  650 = 'Clamp Cylinder A1 Failed to Advance... Check Q1.0...' | German: 'S5 650 Row 66 Failed To Advance.. Check Qxxx.x German' | French: 'S5 650 Row 66 Failed To Advance.. Check Qxxx.x French'
  651 = 'Clamp Cylinder A1 Failed to Return... Check Q1.1...' | German: 'S5 651 Row 66 Failed To Return.. Check Qxxx.x German' | French: 'S5 651 Row 66 Failed To Return.. Check Qxxx.x French'
  652 = 'Clamp Cylinder A1 Lost Advanced... Check I1.0...' | German: 'S5 652 Row 66 Lost Advance Position... Check Ixxx.x German' | French: 'S5 652 Row 66 Lost Advance Position... Check Ixxx.x French'
  653 = 'Clamp Cylinder A1 Lost Returned... Check I1.1...' | German: 'S5 653 Row 66 Lost Return Position... Check Ixxx.x German' | French: 'S5 653 Row 66 Lost Return Position... Check Ixxx.x French'
  654 = 'Clamp Cylinder A1 Switch Fault... Check I1.0, I1.1...' | German: 'S5 654 Row 66 Switch Fault... Check Ixxx.x / Ixxx.x German' | French: 'S5 654 Row 66 Switch Fault... Check Ixxx.x / Ixxx.x French'
  655 = 'Spare' | German: 'S5 655 Row 66 Spare Message German' | French: 'S5 655 Row 66 Spare Message French'
  656 = 'Spare' | German: 'S5 656 Row 66 Spare Message German' | French: 'S5 656 Row 66 Spare Message French'
  657 = 'Spare' | German: 'S5 657 Row 66 Spare Message German' | French: 'S5 657 Row 66 Spare Message French'
  658 = 'Spare' | German: 'S5 658 Row 66 Spare Message German' | French: 'S5 658 Row 66 Spare Message French'
  659 = 'Spare' | German: 'S5 659 Row 66 Spare Message German' | French: 'S5 659 Row 66 Spare Message French'
  660 = 'Clamp Cylinder A1 Failed to Advance... Check Q1.0...' | German: 'S5 660 Row 67 Failed To Advance.. Check Qxxx.x German' | French: 'S5 660 Row 67 Failed To Advance.. Check Qxxx.x French'
  661 = 'Clamp Cylinder A1 Failed to Return... Check Q1.1...' | German: 'S5 661 Row 67 Failed To Return.. Check Qxxx.x German' | French: 'S5 661 Row 67 Failed To Return.. Check Qxxx.x French'
  662 = 'Clamp Cylinder A1 Lost Advanced... Check I1.0...' | German: 'S5 662 Row 67 Lost Advance Position... Check Ixxx.x German' | French: 'S5 662 Row 67 Lost Advance Position... Check Ixxx.x French'
  663 = 'Clamp Cylinder A1 Lost Returned... Check I1.1...' | German: 'S5 663 Row 67 Lost Return Position... Check Ixxx.x German' | French: 'S5 663 Row 67 Lost Return Position... Check Ixxx.x French'
  664 = 'Clamp Cylinder A1 Switch Fault... Check I1.0, I1.1...' | German: 'S5 664 Row 67 Switch Fault... Check Ixxx.x / Ixxx.x German' | French: 'S5 664 Row 67 Switch Fault... Check Ixxx.x / Ixxx.x French'
  665 = 'Spare' | German: 'S5 665 Row 67 Spare Message German' | French: 'S5 665 Row 67 Spare Message French'
  666 = 'Spare' | German: 'S5 666 Row 67 Spare Message German' | French: 'S5 666 Row 67 Spare Message French'
  667 = 'Spare' | German: 'S5 667 Row 67 Spare Message German' | French: 'S5 667 Row 67 Spare Message French'
  668 = 'Spare' | German: 'S5 668 Row 67 Spare Message German' | French: 'S5 668 Row 67 Spare Message French'
  669 = 'Spare' | German: 'S5 669 Row 67 Spare Message German' | French: 'S5 669 Row 67 Spare Message French'
  670 = 'Clamp Cylinder A1 Failed to Advance... Check Q1.0...' | German: 'S5 670 Row 68 Failed To Advance.. Check Qxxx.x German' | French: 'S5 670 Row 68 Failed To Advance.. Check Qxxx.x French'
  671 = 'Clamp Cylinder A1 Failed to Return... Check Q1.1...' | German: 'S5 671 Row 68 Failed To Return.. Check Qxxx.x German' | French: 'S5 671 Row 68 Failed To Return.. Check Qxxx.x French'
  672 = 'Clamp Cylinder A1 Lost Advanced... Check I1.0...' | German: 'S5 672 Row 68 Lost Advance Position... Check Ixxx.x German' | French: 'S5 672 Row 68 Lost Advance Position... Check Ixxx.x French'
  673 = 'Clamp Cylinder A1 Lost Returned... Check I1.1...' | German: 'S5 673 Row 68 Lost Return Position... Check Ixxx.x German' | French: 'S5 673 Row 68 Lost Return Position... Check Ixxx.x French'
  674 = 'Clamp Cylinder A1 Switch Fault... Check I1.0, I1.1...' | German: 'S5 674 Row 68 Switch Fault... Check Ixxx.x / Ixxx.x German' | French: 'S5 674 Row 68 Switch Fault... Check Ixxx.x / Ixxx.x French'
  675 = 'Spare' | German: 'S5 675 Row 68 Spare Message German' | French: 'S5 675 Row 68 Spare Message French'
  676 = 'Spare' | German: 'S5 676 Row 68 Spare Message German' | French: 'S5 676 Row 68 Spare Message French'
  677 = 'Spare' | German: 'S5 677 Row 68 Spare Message German' | French: 'S5 677 Row 68 Spare Message French'
  678 = 'Spare' | German: 'S5 678 Row 68 Spare Message German' | French: 'S5 678 Row 68 Spare Message French'
  679 = 'Spare' | German: 'S5 679 Row 68 Spare Message German' | French: 'S5 679 Row 68 Spare Message French'
  680 = 'Clamp Cylinder A1 Failed to Advance... Check Q1.0...' | German: 'S5 680 Row 69 Failed To Advance.. Check Qxxx.x German' | French: 'S5 680 Row 69 Failed To Advance.. Check Qxxx.x French'
  681 = 'Clamp Cylinder A1 Failed to Return... Check Q1.1...' | German: 'S5 681 Row 69 Failed To Return.. Check Qxxx.x German' | French: 'S5 681 Row 69 Failed To Return.. Check Qxxx.x French'
  682 = 'Clamp Cylinder A1 Lost Advanced... Check I1.0...' | German: 'S5 682 Row 69 Lost Advance Position... Check Ixxx.x German' | French: 'S5 682 Row 69 Lost Advance Position... Check Ixxx.x French'
  683 = 'Clamp Cylinder A1 Lost Returned... Check I1.1...' | German: 'S5 683 Row 69 Lost Return Position... Check Ixxx.x German' | French: 'S5 683 Row 69 Lost Return Position... Check Ixxx.x French'
  684 = 'Clamp Cylinder A1 Switch Fault... Check I1.0, I1.1...' | German: 'S5 684 Row 69 Switch Fault... Check Ixxx.x / Ixxx.x German' | French: 'S5 684 Row 69 Switch Fault... Check Ixxx.x / Ixxx.x French'
  685 = 'Spare' | German: 'S5 685 Row 69 Spare Message German' | French: 'S5 685 Row 69 Spare Message French'
  686 = 'Spare' | German: 'S5 686 Row 69 Spare Message German' | French: 'S5 686 Row 69 Spare Message French'
  687 = 'Spare' | German: 'S5 687 Row 69 Spare Message German' | French: 'S5 687 Row 69 Spare Message French'
  688 = 'Spare' | German: 'S5 688 Row 69 Spare Message German' | French: 'S5 688 Row 69 Spare Message French'
  689 = 'Spare' | German: 'S5 689 Row 69 Spare Message German' | French: 'S5 689 Row 69 Spare Message French'
  690 = 'Clamp Cylinder A1 Failed to Advance... Check Q1.0...' | German: 'S5 690 Row 70 Failed To Advance.. Check Qxxx.x German' | French: 'S5 690 Row 70 Failed To Advance.. Check Qxxx.x French'
  691 = 'Clamp Cylinder A1 Failed to Return... Check Q1.1...' | German: 'S5 691 Row 70 Failed To Return.. Check Qxxx.x German' | French: 'S5 691 Row 70 Failed To Return.. Check Qxxx.x French'
  692 = 'Clamp Cylinder A1 Lost Advanced... Check I1.0...' | German: 'S5 692 Row 70 Lost Advance Position... Check Ixxx.x German' | French: 'S5 692 Row 70 Lost Advance Position... Check Ixxx.x French'
  693 = 'Clamp Cylinder A1 Lost Returned... Check I1.1...' | German: 'S5 693 Row 70 Lost Return Position... Check Ixxx.x German' | French: 'S5 693 Row 70 Lost Return Position... Check Ixxx.x French'
  694 = 'Clamp Cylinder A1 Switch Fault... Check I1.0, I1.1...' | German: 'S5 694 Row 70 Switch Fault... Check Ixxx.x / Ixxx.x German' | French: 'S5 694 Row 70 Switch Fault... Check Ixxx.x / Ixxx.x French'
  695 = 'Spare' | German: 'S5 695 Row 70 Spare Message German' | French: 'S5 695 Row 70 Spare Message French'
  696 = 'Spare' | German: 'S5 696 Row 70 Spare Message German' | French: 'S5 696 Row 70 Spare Message French'
  697 = 'Spare' | German: 'S5 697 Row 70 Spare Message German' | French: 'S5 697 Row 70 Spare Message French'
  698 = 'Spare' | German: 'S5 698 Row 70 Spare Message German' | French: 'S5 698 Row 70 Spare Message French'
  699 = 'Spare' | German: 'S5 699 Row 70 Spare Message German' | French: 'S5 699 Row 70 Spare Message French'
  700 = 'Clamp Cylinder A1 Failed to Advance... Check Q1.0...' | German: 'S5 700 Row 71 Failed To Advance.. Check Qxxx.x German' | French: 'S5 700 Row 71 Failed To Advance.. Check Qxxx.x French'
  701 = 'Clamp Cylinder A1 Failed to Return... Check Q1.1...' | German: 'S5 701 Row 71 Failed To Return.. Check Qxxx.x German' | French: 'S5 701 Row 71 Failed To Return.. Check Qxxx.x French'
  702 = 'Clamp Cylinder A1 Lost Advanced... Check I1.0...' | German: 'S5 702 Row 71 Lost Advance Position... Check Ixxx.x German' | French: 'S5 702 Row 71 Lost Advance Position... Check Ixxx.x French'
  703 = 'Clamp Cylinder A1 Lost Returned... Check I1.1...' | German: 'S5 703 Row 71 Lost Return Position... Check Ixxx.x German' | French: 'S5 703 Row 71 Lost Return Position... Check Ixxx.x French'
  704 = 'Clamp Cylinder A1 Switch Fault... Check I1.0, I1.1...' | German: 'S5 704 Row 71 Switch Fault... Check Ixxx.x / Ixxx.x German' | French: 'S5 704 Row 71 Switch Fault... Check Ixxx.x / Ixxx.x French'
  705 = 'Spare' | German: 'S5 705 Row 71 Spare Message German' | French: 'S5 705 Row 71 Spare Message French'
  706 = 'Spare' | German: 'S5 706 Row 71 Spare Message German' | French: 'S5 706 Row 71 Spare Message French'
  707 = 'Spare' | German: 'S5 707 Row 71 Spare Message German' | French: 'S5 707 Row 71 Spare Message French'
  708 = 'Spare' | German: 'S5 708 Row 71 Spare Message German' | French: 'S5 708 Row 71 Spare Message French'
  709 = 'Spare' | German: 'S5 709 Row 71 Spare Message German' | French: 'S5 709 Row 71 Spare Message French'
  710 = 'Clamp Cylinder A1 Failed to Advance... Check Q1.0...' | German: 'S5 710 Row 72 Failed To Advance.. Check Qxxx.x German' | French: 'S5 710 Row 72 Failed To Advance.. Check Qxxx.x French'
  711 = 'Clamp Cylinder A1 Failed to Return... Check Q1.1...' | German: 'S5 711 Row 72 Failed To Return.. Check Qxxx.x German' | French: 'S5 711 Row 72 Failed To Return.. Check Qxxx.x French'
  712 = 'Clamp Cylinder A1 Lost Advanced... Check I1.0...' | German: 'S5 712 Row 72 Lost Advance Position... Check Ixxx.x German' | French: 'S5 712 Row 72 Lost Advance Position... Check Ixxx.x French'
  713 = 'Clamp Cylinder A1 Lost Returned... Check I1.1...' | German: 'S5 713 Row 72 Lost Return Position... Check Ixxx.x German' | French: 'S5 713 Row 72 Lost Return Position... Check Ixxx.x French'
  714 = 'Clamp Cylinder A1 Switch Fault... Check I1.0, I1.1...' | German: 'S5 714 Row 72 Switch Fault... Check Ixxx.x / Ixxx.x German' | French: 'S5 714 Row 72 Switch Fault... Check Ixxx.x / Ixxx.x French'
  715 = 'Spare' | German: 'S5 715 Row 72 Spare Message German' | French: 'S5 715 Row 72 Spare Message French'
  716 = 'Spare' | German: 'S5 716 Row 72 Spare Message German' | French: 'S5 716 Row 72 Spare Message French'
  717 = 'Spare' | German: 'S5 717 Row 72 Spare Message German' | French: 'S5 717 Row 72 Spare Message French'
  718 = 'Spare' | German: 'S5 718 Row 72 Spare Message German' | French: 'S5 718 Row 72 Spare Message French'
  719 = 'Spare' | German: 'S5 719 Row 72 Spare Message German' | French: 'S5 719 Row 72 Spare Message French'
  720 = 'Clamp Cylinder A1 Failed to Advance... Check Q1.0...' | German: 'S5 720 Row 73 Failed To Advance.. Check Qxxx.x German' | French: 'S5 720 Row 73 Failed To Advance.. Check Qxxx.x French'
  721 = 'Clamp Cylinder A1 Failed to Return... Check Q1.1...' | German: 'S5 721 Row 73 Failed To Return.. Check Qxxx.x German' | French: 'S5 721 Row 73 Failed To Return.. Check Qxxx.x French'
  722 = 'Clamp Cylinder A1 Lost Advanced... Check I1.0...' | German: 'S5 722 Row 73 Lost Advance Position... Check Ixxx.x German' | French: 'S5 722 Row 73 Lost Advance Position... Check Ixxx.x French'
  723 = 'Clamp Cylinder A1 Lost Returned... Check I1.1...' | German: 'S5 723 Row 73 Lost Return Position... Check Ixxx.x German' | French: 'S5 723 Row 73 Lost Return Position... Check Ixxx.x French'
  724 = 'Clamp Cylinder A1 Switch Fault... Check I1.0, I1.1...' | German: 'S5 724 Row 73 Switch Fault... Check Ixxx.x / Ixxx.x German' | French: 'S5 724 Row 73 Switch Fault... Check Ixxx.x / Ixxx.x French'
  725 = 'Spare' | German: 'S5 725 Row 73 Spare Message German' | French: 'S5 725 Row 73 Spare Message French'
  726 = 'Spare' | German: 'S5 726 Row 73 Spare Message German' | French: 'S5 726 Row 73 Spare Message French'
  727 = 'Spare' | German: 'S5 727 Row 73 Spare Message German' | French: 'S5 727 Row 73 Spare Message French'
  728 = 'Spare' | German: 'S5 728 Row 73 Spare Message German' | French: 'S5 728 Row 73 Spare Message French'
  729 = 'Spare' | German: 'S5 729 Row 73 Spare Message German' | French: 'S5 729 Row 73 Spare Message French'
  730 = 'Clamp Cylinder A1 Failed to Advance... Check Q1.0...' | German: 'S5 730 Row 74 Failed To Advance.. Check Qxxx.x German' | French: 'S5 730 Row 74 Failed To Advance.. Check Qxxx.x French'
  731 = 'Clamp Cylinder A1 Failed to Return... Check Q1.1...' | German: 'S5 731 Row 74 Failed To Return.. Check Qxxx.x German' | French: 'S5 731 Row 74 Failed To Return.. Check Qxxx.x French'
  732 = 'Clamp Cylinder A1 Lost Advanced... Check I1.0...' | German: 'S5 732 Row 74 Lost Advance Position... Check Ixxx.x German' | French: 'S5 732 Row 74 Lost Advance Position... Check Ixxx.x French'
  733 = 'Clamp Cylinder A1 Lost Returned... Check I1.1...' | German: 'S5 733 Row 74 Lost Return Position... Check Ixxx.x German' | French: 'S5 733 Row 74 Lost Return Position... Check Ixxx.x French'
  734 = 'Clamp Cylinder A1 Switch Fault... Check I1.0, I1.1...' | German: 'S5 734 Row 74 Switch Fault... Check Ixxx.x / Ixxx.x German' | French: 'S5 734 Row 74 Switch Fault... Check Ixxx.x / Ixxx.x French'
  735 = 'Spare' | German: 'S5 735 Row 74 Spare Message German' | French: 'S5 735 Row 74 Spare Message French'
  736 = 'Spare' | German: 'S5 736 Row 74 Spare Message German' | French: 'S5 736 Row 74 Spare Message French'
  737 = 'Spare' | German: 'S5 737 Row 74 Spare Message German' | French: 'S5 737 Row 74 Spare Message French'
  738 = 'Spare' | German: 'S5 738 Row 74 Spare Message German' | French: 'S5 738 Row 74 Spare Message French'
  739 = 'Spare' | German: 'S5 739 Row 74 Spare Message German' | French: 'S5 739 Row 74 Spare Message French'
  740 = 'Clamp Cylinder A1 Failed to Advance... Check Q1.0...' | German: 'S5 740 Row 75 Failed To Advance.. Check Qxxx.x German' | French: 'S5 740 Row 75 Failed To Advance.. Check Qxxx.x French'
  741 = 'Clamp Cylinder A1 Failed to Return... Check Q1.1...' | German: 'S5 741 Row 75 Failed To Return.. Check Qxxx.x German' | French: 'S5 741 Row 75 Failed To Return.. Check Qxxx.x French'
  742 = 'Clamp Cylinder A1 Lost Advanced... Check I1.0...' | German: 'S5 742 Row 75 Lost Advance Position... Check Ixxx.x German' | French: 'S5 742 Row 75 Lost Advance Position... Check Ixxx.x French'
  743 = 'Clamp Cylinder A1 Lost Returned... Check I1.1...' | German: 'S5 743 Row 75 Lost Return Position... Check Ixxx.x German' | French: 'S5 743 Row 75 Lost Return Position... Check Ixxx.x French'
  744 = 'Clamp Cylinder A1 Switch Fault... Check I1.0, I1.1...' | German: 'S5 744 Row 75 Switch Fault... Check Ixxx.x / Ixxx.x German' | French: 'S5 744 Row 75 Switch Fault... Check Ixxx.x / Ixxx.x French'
  745 = 'Spare' | German: 'S5 745 Row 75 Spare Message German' | French: 'S5 745 Row 75 Spare Message French'
  746 = 'Spare' | German: 'S5 746 Row 75 Spare Message German' | French: 'S5 746 Row 75 Spare Message French'
  747 = 'Spare' | German: 'S5 747 Row 75 Spare Message German' | French: 'S5 747 Row 75 Spare Message French'
  748 = 'Spare' | German: 'S5 748 Row 75 Spare Message German' | French: 'S5 748 Row 75 Spare Message French'
  749 = 'Spare' | German: 'S5 749 Row 75 Spare Message German' | French: 'S5 749 Row 75 Spare Message French'
  750 = 'Clamp Cylinder A1 Failed to Advance... Check Q1.0...' | German: 'S5 750 Row 76 Failed To Advance.. Check Qxxx.x German' | French: 'S5 750 Row 76 Failed To Advance.. Check Qxxx.x French'
  751 = 'Clamp Cylinder A1 Failed to Return... Check Q1.1...' | German: 'S5 751 Row 76 Failed To Return.. Check Qxxx.x German' | French: 'S5 751 Row 76 Failed To Return.. Check Qxxx.x French'
  752 = 'Clamp Cylinder A1 Lost Advanced... Check I1.0...' | German: 'S5 752 Row 76 Lost Advance Position... Check Ixxx.x German' | French: 'S5 752 Row 76 Lost Advance Position... Check Ixxx.x French'
  753 = 'Clamp Cylinder A1 Lost Returned... Check I1.1...' | German: 'S5 753 Row 76 Lost Return Position... Check Ixxx.x German' | French: 'S5 753 Row 76 Lost Return Position... Check Ixxx.x French'
  754 = 'Clamp Cylinder A1 Switch Fault... Check I1.0, I1.1...' | German: 'S5 754 Row 76 Switch Fault... Check Ixxx.x / Ixxx.x German' | French: 'S5 754 Row 76 Switch Fault... Check Ixxx.x / Ixxx.x French'
  755 = 'Spare' | German: 'S5 755 Row 76 Spare Message German' | French: 'S5 755 Row 76 Spare Message French'
  756 = 'Spare' | German: 'S5 756 Row 76 Spare Message German' | French: 'S5 756 Row 76 Spare Message French'
  757 = 'Spare' | German: 'S5 757 Row 76 Spare Message German' | French: 'S5 757 Row 76 Spare Message French'
  758 = 'Spare' | German: 'S5 758 Row 76 Spare Message German' | French: 'S5 758 Row 76 Spare Message French'
  759 = 'Spare' | German: 'S5 759 Row 76 Spare Message German' | French: 'S5 759 Row 76 Spare Message French'
  760 = 'Clamp Cylinder A1 Failed to Advance... Check Q1.0...' | German: 'S5 760 Row 77 Failed To Advance.. Check Qxxx.x German' | French: 'S5 760 Row 77 Failed To Advance.. Check Qxxx.x French'
  761 = 'Clamp Cylinder A1 Failed to Return... Check Q1.1...' | German: 'S5 761 Row 77 Failed To Return.. Check Qxxx.x German' | French: 'S5 761 Row 77 Failed To Return.. Check Qxxx.x French'
  762 = 'Clamp Cylinder A1 Lost Advanced... Check I1.0...' | German: 'S5 762 Row 77 Lost Advance Position... Check Ixxx.x German' | French: 'S5 762 Row 77 Lost Advance Position... Check Ixxx.x French'
  763 = 'Clamp Cylinder A1 Lost Returned... Check I1.1...' | German: 'S5 763 Row 77 Lost Return Position... Check Ixxx.x German' | French: 'S5 763 Row 77 Lost Return Position... Check Ixxx.x French'
  764 = 'Clamp Cylinder A1 Switch Fault... Check I1.0, I1.1...' | German: 'S5 764 Row 77 Switch Fault... Check Ixxx.x / Ixxx.x German' | French: 'S5 764 Row 77 Switch Fault... Check Ixxx.x / Ixxx.x French'
  765 = 'Spare' | German: 'S5 765 Row 77 Spare Message German' | French: 'S5 765 Row 77 Spare Message French'
  766 = 'Spare' | German: 'S5 766 Row 77 Spare Message German' | French: 'S5 766 Row 77 Spare Message French'
  767 = 'Spare' | German: 'S5 767 Row 77 Spare Message German' | French: 'S5 767 Row 77 Spare Message French'
  768 = 'Spare' | German: 'S5 768 Row 77 Spare Message German' | French: 'S5 768 Row 77 Spare Message French'
  769 = 'Spare' | German: 'S5 769 Row 77 Spare Message German' | French: 'S5 769 Row 77 Spare Message French'
  770 = 'Clamp Cylinder A1 Failed to Advance... Check Q1.0...' | German: 'S5 770 Row 78 Failed To Advance.. Check Qxxx.x German' | French: 'S5 770 Row 78 Failed To Advance.. Check Qxxx.x French'
  771 = 'Clamp Cylinder A1 Failed to Return... Check Q1.1...' | German: 'S5 771 Row 78 Failed To Return.. Check Qxxx.x German' | French: 'S5 771 Row 78 Failed To Return.. Check Qxxx.x French'
  772 = 'Clamp Cylinder A1 Lost Advanced... Check I1.0...' | German: 'S5 772 Row 78 Lost Advance Position... Check Ixxx.x German' | French: 'S5 772 Row 78 Lost Advance Position... Check Ixxx.x French'
  773 = 'Clamp Cylinder A1 Lost Returned... Check I1.1...' | German: 'S5 773 Row 78 Lost Return Position... Check Ixxx.x German' | French: 'S5 773 Row 78 Lost Return Position... Check Ixxx.x French'
  774 = 'Clamp Cylinder A1 Switch Fault... Check I1.0, I1.1...' | German: 'S5 774 Row 78 Switch Fault... Check Ixxx.x / Ixxx.x German' | French: 'S5 774 Row 78 Switch Fault... Check Ixxx.x / Ixxx.x French'
  775 = 'Spare' | German: 'S5 775 Row 78 Spare Message German' | French: 'S5 775 Row 78 Spare Message French'
  776 = 'Spare' | German: 'S5 776 Row 78 Spare Message German' | French: 'S5 776 Row 78 Spare Message French'
  777 = 'Spare' | German: 'S5 777 Row 78 Spare Message German' | French: 'S5 777 Row 78 Spare Message French'
  778 = 'Spare' | German: 'S5 778 Row 78 Spare Message German' | French: 'S5 778 Row 78 Spare Message French'
  779 = 'Spare' | German: 'S5 779 Row 78 Spare Message German' | French: 'S5 779 Row 78 Spare Message French'
  780 = 'Clamp Cylinder A1 Failed to Advance... Check Q1.0...' | German: 'S5 780 Row 79 Failed To Advance.. Check Qxxx.x German' | French: 'S5 780 Row 79 Failed To Advance.. Check Qxxx.x French'
  781 = 'Clamp Cylinder A1 Failed to Return... Check Q1.1...' | German: 'S5 781 Row 79 Failed To Return.. Check Qxxx.x German' | French: 'S5 781 Row 79 Failed To Return.. Check Qxxx.x French'
  782 = 'Clamp Cylinder A1 Lost Advanced... Check I1.0...' | German: 'S5 782 Row 79 Lost Advance Position... Check Ixxx.x German' | French: 'S5 782 Row 79 Lost Advance Position... Check Ixxx.x French'
  783 = 'Clamp Cylinder A1 Lost Returned... Check I1.1...' | German: 'S5 783 Row 79 Lost Return Position... Check Ixxx.x German' | French: 'S5 783 Row 79 Lost Return Position... Check Ixxx.x French'
  784 = 'Clamp Cylinder A1 Switch Fault... Check I1.0, I1.1...' | German: 'S5 784 Row 79 Switch Fault... Check Ixxx.x / Ixxx.x German' | French: 'S5 784 Row 79 Switch Fault... Check Ixxx.x / Ixxx.x French'
  785 = 'Spare' | German: 'S5 785 Row 79 Spare Message German' | French: 'S5 785 Row 79 Spare Message French'
  786 = 'Spare' | German: 'S5 786 Row 79 Spare Message German' | French: 'S5 786 Row 79 Spare Message French'
  787 = 'Spare' | German: 'S5 787 Row 79 Spare Message German' | French: 'S5 787 Row 79 Spare Message French'
  788 = 'Spare' | German: 'S5 788 Row 79 Spare Message German' | French: 'S5 788 Row 79 Spare Message French'
  789 = 'Spare' | German: 'S5 789 Row 79 Spare Message German' | French: 'S5 789 Row 79 Spare Message French'
  790 = 'Clamp Cylinder A1 Failed to Advance... Check Q1.0...' | German: 'S5 790 Row 80 Failed To Advance.. Check Qxxx.x German' | French: 'S5 790 Row 80 Failed To Advance.. Check Qxxx.x French'
  791 = 'Clamp Cylinder A1 Failed to Return... Check Q1.1...' | German: 'S5 791 Row 80 Failed To Return.. Check Qxxx.x German' | French: 'S5 791 Row 80 Failed To Return.. Check Qxxx.x French'
  792 = 'Clamp Cylinder A1 Lost Advanced... Check I1.0...' | German: 'S5 792 Row 80 Lost Advance Position... Check Ixxx.x German' | French: 'S5 792 Row 80 Lost Advance Position... Check Ixxx.x French'
  793 = 'Clamp Cylinder A1 Lost Returned... Check I1.1...' | German: 'S5 793 Row 80 Lost Return Position... Check Ixxx.x German' | French: 'S5 793 Row 80 Lost Return Position... Check Ixxx.x French'
  794 = 'Clamp Cylinder A1 Switch Fault... Check I1.0, I1.1...' | German: 'S5 794 Row 80 Switch Fault... Check Ixxx.x / Ixxx.x German' | French: 'S5 794 Row 80 Switch Fault... Check Ixxx.x / Ixxx.x French'
  795 = 'Spare' | German: 'S5 795 Row 80 Spare Message German' | French: 'S5 795 Row 80 Spare Message French'
  796 = 'Spare' | German: 'S5 796 Row 80 Spare Message German' | French: 'S5 796 Row 80 Spare Message French'
  797 = 'Spare' | German: 'S5 797 Row 80 Spare Message German' | French: 'S5 797 Row 80 Spare Message French'
  798 = 'Spare' | German: 'S5 798 Row 80 Spare Message German' | French: 'S5 798 Row 80 Spare Message French'
  799 = 'Spare' | German: 'S5 799 Row 80 Spare Message German' | French: 'S5 799 Row 80 Spare Message French'
  800 = 'Clamp Cylinder A1 Failed to Advance... Check Q1.0...' | German: 'S5 800 Row 81 Failed To Advance.. Check Qxxx.x German' | French: 'S5 800 Row 81 Failed To Advance.. Check Qxxx.x French'
  801 = 'Clamp Cylinder A1 Failed to Return... Check Q1.1...' | German: 'S5 801 Row 81 Failed To Return.. Check Qxxx.x German' | French: 'S5 801 Row 81 Failed To Return.. Check Qxxx.x French'
  802 = 'Clamp Cylinder A1 Lost Advanced... Check I1.0...' | German: 'S5 802 Row 81 Lost Advance Position... Check Ixxx.x German' | French: 'S5 802 Row 81 Lost Advance Position... Check Ixxx.x French'
  803 = 'Clamp Cylinder A1 Lost Returned... Check I1.1...' | German: 'S5 803 Row 81 Lost Return Position... Check Ixxx.x German' | French: 'S5 803 Row 81 Lost Return Position... Check Ixxx.x French'
  804 = 'Clamp Cylinder A1 Switch Fault... Check I1.0, I1.1...' | German: 'S5 804 Row 81 Switch Fault... Check Ixxx.x / Ixxx.x German' | French: 'S5 804 Row 81 Switch Fault... Check Ixxx.x / Ixxx.x French'
  805 = 'Spare' | German: 'S5 805 Row 81 Spare Message German' | French: 'S5 805 Row 81 Spare Message French'
  806 = 'Spare' | German: 'S5 806 Row 81 Spare Message German' | French: 'S5 806 Row 81 Spare Message French'
  807 = 'Spare' | German: 'S5 807 Row 81 Spare Message German' | French: 'S5 807 Row 81 Spare Message French'
  808 = 'Spare' | German: 'S5 808 Row 81 Spare Message German' | French: 'S5 808 Row 81 Spare Message French'
  809 = 'Spare' | German: 'S5 809 Row 81 Spare Message German' | French: 'S5 809 Row 81 Spare Message French'
  810 = 'Clamp Cylinder A1 Failed to Advance... Check Q1.0...' | German: 'S5 810 Row 82 Failed To Advance.. Check Qxxx.x German' | French: 'S5 810 Row 82 Failed To Advance.. Check Qxxx.x French'
  811 = 'Clamp Cylinder A1 Failed to Return... Check Q1.1...' | German: 'S5 811 Row 82 Failed To Return.. Check Qxxx.x German' | French: 'S5 811 Row 82 Failed To Return.. Check Qxxx.x French'
  812 = 'Clamp Cylinder A1 Lost Advanced... Check I1.0...' | German: 'S5 812 Row 82 Lost Advance Position... Check Ixxx.x German' | French: 'S5 812 Row 82 Lost Advance Position... Check Ixxx.x French'
  813 = 'Clamp Cylinder A1 Lost Returned... Check I1.1...' | German: 'S5 813 Row 82 Lost Return Position... Check Ixxx.x German' | French: 'S5 813 Row 82 Lost Return Position... Check Ixxx.x French'
  814 = 'Clamp Cylinder A1 Switch Fault... Check I1.0, I1.1...' | German: 'S5 814 Row 82 Switch Fault... Check Ixxx.x / Ixxx.x German' | French: 'S5 814 Row 82 Switch Fault... Check Ixxx.x / Ixxx.x French'
  815 = 'Spare' | German: 'S5 815 Row 82 Spare Message German' | French: 'S5 815 Row 82 Spare Message French'
  816 = 'Spare' | German: 'S5 816 Row 82 Spare Message German' | French: 'S5 816 Row 82 Spare Message French'
  817 = 'Spare' | German: 'S5 817 Row 82 Spare Message German' | French: 'S5 817 Row 82 Spare Message French'
  818 = 'Spare' | German: 'S5 818 Row 82 Spare Message German' | French: 'S5 818 Row 82 Spare Message French'
  819 = 'Spare' | German: 'S5 819 Row 82 Spare Message German' | French: 'S5 819 Row 82 Spare Message French'
  820 = 'Clamp Cylinder A1 Failed to Advance... Check Q1.0...' | German: 'S5 820 Row 83 Failed To Advance.. Check Qxxx.x German' | French: 'S5 820 Row 83 Failed To Advance.. Check Qxxx.x French'
  821 = 'Clamp Cylinder A1 Failed to Return... Check Q1.1...' | German: 'S5 821 Row 83 Failed To Return.. Check Qxxx.x German' | French: 'S5 821 Row 83 Failed To Return.. Check Qxxx.x French'
  822 = 'Clamp Cylinder A1 Lost Advanced... Check I1.0...' | German: 'S5 822 Row 83 Lost Advance Position... Check Ixxx.x German' | French: 'S5 822 Row 83 Lost Advance Position... Check Ixxx.x French'
  823 = 'Clamp Cylinder A1 Lost Returned... Check I1.1...' | German: 'S5 823 Row 83 Lost Return Position... Check Ixxx.x German' | French: 'S5 823 Row 83 Lost Return Position... Check Ixxx.x French'
  824 = 'Clamp Cylinder A1 Switch Fault... Check I1.0, I1.1...' | German: 'S5 824 Row 83 Switch Fault... Check Ixxx.x / Ixxx.x German' | French: 'S5 824 Row 83 Switch Fault... Check Ixxx.x / Ixxx.x French'
  825 = 'Spare' | German: 'S5 825 Row 83 Spare Message German' | French: 'S5 825 Row 83 Spare Message French'
  826 = 'Spare' | German: 'S5 826 Row 83 Spare Message German' | French: 'S5 826 Row 83 Spare Message French'
  827 = 'Spare' | German: 'S5 827 Row 83 Spare Message German' | French: 'S5 827 Row 83 Spare Message French'
  828 = 'Spare' | German: 'S5 828 Row 83 Spare Message German' | French: 'S5 828 Row 83 Spare Message French'
  829 = 'Spare' | German: 'S5 829 Row 83 Spare Message German' | French: 'S5 829 Row 83 Spare Message French'
  830 = 'Clamp Cylinder A1 Failed to Advance... Check Q1.0...' | German: 'S5 830 Row 84 Failed To Advance.. Check Qxxx.x German' | French: 'S5 830 Row 84 Failed To Advance.. Check Qxxx.x French'
  831 = 'Clamp Cylinder A1 Failed to Return... Check Q1.1...' | German: 'S5 831 Row 84 Failed To Return.. Check Qxxx.x German' | French: 'S5 831 Row 84 Failed To Return.. Check Qxxx.x French'
  832 = 'Clamp Cylinder A1 Lost Advanced... Check I1.0...' | German: 'S5 832 Row 84 Lost Advance Position... Check Ixxx.x German' | French: 'S5 832 Row 84 Lost Advance Position... Check Ixxx.x French'
  833 = 'Clamp Cylinder A1 Lost Returned... Check I1.1...' | German: 'S5 833 Row 84 Lost Return Position... Check Ixxx.x German' | French: 'S5 833 Row 84 Lost Return Position... Check Ixxx.x French'
  834 = 'Clamp Cylinder A1 Switch Fault... Check I1.0, I1.1...' | German: 'S5 834 Row 84 Switch Fault... Check Ixxx.x / Ixxx.x German' | French: 'S5 834 Row 84 Switch Fault... Check Ixxx.x / Ixxx.x French'
  835 = 'Spare' | German: 'S5 835 Row 84 Spare Message German' | French: 'S5 835 Row 84 Spare Message French'
  836 = 'Spare' | German: 'S5 836 Row 84 Spare Message German' | French: 'S5 836 Row 84 Spare Message French'
  837 = 'Spare' | German: 'S5 837 Row 84 Spare Message German' | French: 'S5 837 Row 84 Spare Message French'
  838 = 'Spare' | German: 'S5 838 Row 84 Spare Message German' | French: 'S5 838 Row 84 Spare Message French'
  839 = 'Spare' | German: 'S5 839 Row 84 Spare Message German' | French: 'S5 839 Row 84 Spare Message French'
  840 = 'Clamp Cylinder A1 Failed to Advance... Check Q1.0...' | German: 'S5 840 Row 85 Failed To Advance.. Check Qxxx.x German' | French: 'S5 840 Row 85 Failed To Advance.. Check Qxxx.x French'
  841 = 'Clamp Cylinder A1 Failed to Return... Check Q1.1...' | German: 'S5 841 Row 85 Failed To Return.. Check Qxxx.x German' | French: 'S5 841 Row 85 Failed To Return.. Check Qxxx.x French'
  842 = 'Clamp Cylinder A1 Lost Advanced... Check I1.0...' | German: 'S5 842 Row 85 Lost Advance Position... Check Ixxx.x German' | French: 'S5 842 Row 85 Lost Advance Position... Check Ixxx.x French'
  843 = 'Clamp Cylinder A1 Lost Returned... Check I1.1...' | German: 'S5 843 Row 85 Lost Return Position... Check Ixxx.x German' | French: 'S5 843 Row 85 Lost Return Position... Check Ixxx.x French'
  844 = 'Clamp Cylinder A1 Switch Fault... Check I1.0, I1.1...' | German: 'S5 844 Row 85 Switch Fault... Check Ixxx.x / Ixxx.x German' | French: 'S5 844 Row 85 Switch Fault... Check Ixxx.x / Ixxx.x French'
  845 = 'Spare' | German: 'S5 845 Row 85 Spare Message German' | French: 'S5 845 Row 85 Spare Message French'
  846 = 'Spare' | German: 'S5 846 Row 85 Spare Message German' | French: 'S5 846 Row 85 Spare Message French'
  847 = 'Spare' | German: 'S5 847 Row 85 Spare Message German' | French: 'S5 847 Row 85 Spare Message French'
  848 = 'Spare' | German: 'S5 848 Row 85 Spare Message German' | French: 'S5 848 Row 85 Spare Message French'
  849 = 'Spare' | German: 'S5 849 Row 85 Spare Message German' | French: 'S5 849 Row 85 Spare Message French'
  850 = 'Clamp Cylinder A1 Failed to Advance... Check Q1.0...' | German: 'S5 850 Row 86 Failed To Advance.. Check Qxxx.x German' | French: 'S5 850 Row 86 Failed To Advance.. Check Qxxx.x French'
  851 = 'Clamp Cylinder A1 Failed to Return... Check Q1.1...' | German: 'S5 851 Row 86 Failed To Return.. Check Qxxx.x German' | French: 'S5 851 Row 86 Failed To Return.. Check Qxxx.x French'
  852 = 'Clamp Cylinder A1 Lost Advanced... Check I1.0...' | German: 'S5 852 Row 86 Lost Advance Position... Check Ixxx.x German' | French: 'S5 852 Row 86 Lost Advance Position... Check Ixxx.x French'
  853 = 'Clamp Cylinder A1 Lost Returned... Check I1.1...' | German: 'S5 853 Row 86 Lost Return Position... Check Ixxx.x German' | French: 'S5 853 Row 86 Lost Return Position... Check Ixxx.x French'
  854 = 'Clamp Cylinder A1 Switch Fault... Check I1.0, I1.1...' | German: 'S5 854 Row 86 Switch Fault... Check Ixxx.x / Ixxx.x German' | French: 'S5 854 Row 86 Switch Fault... Check Ixxx.x / Ixxx.x French'
  855 = 'Spare' | German: 'S5 855 Row 86 Spare Message German' | French: 'S5 855 Row 86 Spare Message French'
  856 = 'Spare' | German: 'S5 856 Row 86 Spare Message German' | French: 'S5 856 Row 86 Spare Message French'
  857 = 'Spare' | German: 'S5 857 Row 86 Spare Message German' | French: 'S5 857 Row 86 Spare Message French'
  858 = 'Spare' | German: 'S5 858 Row 86 Spare Message German' | French: 'S5 858 Row 86 Spare Message French'
  859 = 'Spare' | German: 'S5 859 Row 86 Spare Message German' | French: 'S5 859 Row 86 Spare Message French'
  860 = 'Clamp Cylinder A1 Failed to Advance... Check Q1.0...' | German: 'S5 860 Row 87 Failed To Advance.. Check Qxxx.x German' | French: 'S5 860 Row 87 Failed To Advance.. Check Qxxx.x French'
  861 = 'Clamp Cylinder A1 Failed to Return... Check Q1.1...' | German: 'S5 861 Row 87 Failed To Return.. Check Qxxx.x German' | French: 'S5 861 Row 87 Failed To Return.. Check Qxxx.x French'
  862 = 'Clamp Cylinder A1 Lost Advanced... Check I1.0...' | German: 'S5 862 Row 87 Lost Advance Position... Check Ixxx.x German' | French: 'S5 862 Row 87 Lost Advance Position... Check Ixxx.x French'
  863 = 'Clamp Cylinder A1 Lost Returned... Check I1.1...' | German: 'S5 863 Row 87 Lost Return Position... Check Ixxx.x German' | French: 'S5 863 Row 87 Lost Return Position... Check Ixxx.x French'
  864 = 'Clamp Cylinder A1 Switch Fault... Check I1.0, I1.1...' | German: 'S5 864 Row 87 Switch Fault... Check Ixxx.x / Ixxx.x German' | French: 'S5 864 Row 87 Switch Fault... Check Ixxx.x / Ixxx.x French'
  865 = 'Spare' | German: 'S5 865 Row 87 Spare Message German' | French: 'S5 865 Row 87 Spare Message French'
  866 = 'Spare' | German: 'S5 866 Row 87 Spare Message German' | French: 'S5 866 Row 87 Spare Message French'
  867 = 'Spare' | German: 'S5 867 Row 87 Spare Message German' | French: 'S5 867 Row 87 Spare Message French'
  868 = 'Spare' | German: 'S5 868 Row 87 Spare Message German' | French: 'S5 868 Row 87 Spare Message French'
  869 = 'Spare' | German: 'S5 869 Row 87 Spare Message German' | French: 'S5 869 Row 87 Spare Message French'
  870 = 'Clamp Cylinder A1 Failed to Advance... Check Q1.0...' | German: 'S5 870 Row 88 Failed To Advance.. Check Qxxx.x German' | French: 'S5 870 Row 88 Failed To Advance.. Check Qxxx.x French'
  871 = 'Clamp Cylinder A1 Failed to Return... Check Q1.1...' | German: 'S5 871 Row 88 Failed To Return.. Check Qxxx.x German' | French: 'S5 871 Row 88 Failed To Return.. Check Qxxx.x French'
  872 = 'Clamp Cylinder A1 Lost Advanced... Check I1.0...' | German: 'S5 872 Row 88 Lost Advance Position... Check Ixxx.x German' | French: 'S5 872 Row 88 Lost Advance Position... Check Ixxx.x French'
  873 = 'Clamp Cylinder A1 Lost Returned... Check I1.1...' | German: 'S5 873 Row 88 Lost Return Position... Check Ixxx.x German' | French: 'S5 873 Row 88 Lost Return Position... Check Ixxx.x French'
  874 = 'Clamp Cylinder A1 Switch Fault... Check I1.0, I1.1...' | German: 'S5 874 Row 88 Switch Fault... Check Ixxx.x / Ixxx.x German' | French: 'S5 874 Row 88 Switch Fault... Check Ixxx.x / Ixxx.x French'
  875 = 'Spare' | German: 'S5 875 Row 88 Spare Message German' | French: 'S5 875 Row 88 Spare Message French'
  876 = 'Spare' | German: 'S5 876 Row 88 Spare Message German' | French: 'S5 876 Row 88 Spare Message French'
  877 = 'Spare' | German: 'S5 877 Row 88 Spare Message German' | French: 'S5 877 Row 88 Spare Message French'
  878 = 'Spare' | German: 'S5 878 Row 88 Spare Message German' | French: 'S5 878 Row 88 Spare Message French'
  879 = 'Spare' | German: 'S5 879 Row 88 Spare Message German' | French: 'S5 879 Row 88 Spare Message French'
  880 = 'Clamp Cylinder A1 Failed to Advance... Check Q1.0...' | German: 'S5 880 Row 89 Failed To Advance.. Check Qxxx.x German' | French: 'S5 880 Row 89 Failed To Advance.. Check Qxxx.x French'
  881 = 'Clamp Cylinder A1 Failed to Return... Check Q1.1...' | German: 'S5 881 Row 89 Failed To Return.. Check Qxxx.x German' | French: 'S5 881 Row 89 Failed To Return.. Check Qxxx.x French'
  882 = 'Clamp Cylinder A1 Lost Advanced... Check I1.0...' | German: 'S5 882 Row 89 Lost Advance Position... Check Ixxx.x German' | French: 'S5 882 Row 89 Lost Advance Position... Check Ixxx.x French'
  883 = 'Clamp Cylinder A1 Lost Returned... Check I1.1...' | German: 'S5 883 Row 89 Lost Return Position... Check Ixxx.x German' | French: 'S5 883 Row 89 Lost Return Position... Check Ixxx.x French'
  884 = 'Clamp Cylinder A1 Switch Fault... Check I1.0, I1.1...' | German: 'S5 884 Row 89 Switch Fault... Check Ixxx.x / Ixxx.x German' | French: 'S5 884 Row 89 Switch Fault... Check Ixxx.x / Ixxx.x French'
  885 = 'Spare' | German: 'S5 885 Row 89 Spare Message German' | French: 'S5 885 Row 89 Spare Message French'
  886 = 'Spare' | German: 'S5 886 Row 89 Spare Message German' | French: 'S5 886 Row 89 Spare Message French'
  887 = 'Spare' | German: 'S5 887 Row 89 Spare Message German' | French: 'S5 887 Row 89 Spare Message French'
  888 = 'Spare' | German: 'S5 888 Row 89 Spare Message German' | French: 'S5 888 Row 89 Spare Message French'
  889 = 'Spare' | German: 'S5 889 Row 89 Spare Message German' | French: 'S5 889 Row 89 Spare Message French'
  890 = 'Clamp Cylinder A1 Failed to Advance... Check Q1.0...' | German: 'S5 890 Row 90 Failed To Advance.. Check Qxxx.x German' | French: 'S5 890 Row 90 Failed To Advance.. Check Qxxx.x French'
  891 = 'Clamp Cylinder A1 Failed to Return... Check Q1.1...' | German: 'S5 891 Row 90 Failed To Return.. Check Qxxx.x German' | French: 'S5 891 Row 90 Failed To Return.. Check Qxxx.x French'
  892 = 'Clamp Cylinder A1 Lost Advanced... Check I1.0...' | German: 'S5 892 Row 90 Lost Advance Position... Check Ixxx.x German' | French: 'S5 892 Row 90 Lost Advance Position... Check Ixxx.x French'
  893 = 'Clamp Cylinder A1 Lost Returned... Check I1.1...' | German: 'S5 893 Row 90 Lost Return Position... Check Ixxx.x German' | French: 'S5 893 Row 90 Lost Return Position... Check Ixxx.x French'
  894 = 'Clamp Cylinder A1 Switch Fault... Check I1.0, I1.1...' | German: 'S5 894 Row 90 Switch Fault... Check Ixxx.x / Ixxx.x German' | French: 'S5 894 Row 90 Switch Fault... Check Ixxx.x / Ixxx.x French'
  895 = 'Spare' | German: 'S5 895 Row 90 Spare Message German' | French: 'S5 895 Row 90 Spare Message French'
  896 = 'Spare' | German: 'S5 896 Row 90 Spare Message German' | French: 'S5 896 Row 90 Spare Message French'
  897 = 'Spare' | German: 'S5 897 Row 90 Spare Message German' | French: 'S5 897 Row 90 Spare Message French'
  898 = 'Spare' | German: 'S5 898 Row 90 Spare Message German' | French: 'S5 898 Row 90 Spare Message French'
  899 = 'Spare' | German: 'S5 899 Row 90 Spare Message German' | French: 'S5 899 Row 90 Spare Message French'
  900 = 'Clamp Cylinder A1 Failed to Advance... Check Q1.0...' | German: 'S5 900 Row 91 Failed To Advance.. Check Qxxx.x German' | French: 'S5 900 Row 91 Failed To Advance.. Check Qxxx.x French'
  901 = 'Clamp Cylinder A1 Failed to Return... Check Q1.1...' | German: 'S5 901 Row 91 Failed To Return.. Check Qxxx.x German' | French: 'S5 901 Row 91 Failed To Return.. Check Qxxx.x French'
  902 = 'Clamp Cylinder A1 Lost Advanced... Check I1.0...' | German: 'S5 902 Row 91 Lost Advance Position... Check Ixxx.x German' | French: 'S5 902 Row 91 Lost Advance Position... Check Ixxx.x French'
  903 = 'Clamp Cylinder A1 Lost Returned... Check I1.1...' | German: 'S5 903 Row 91 Lost Return Position... Check Ixxx.x German' | French: 'S5 903 Row 91 Lost Return Position... Check Ixxx.x French'
  904 = 'Clamp Cylinder A1 Switch Fault... Check I1.0, I1.1...' | German: 'S5 904 Row 91 Switch Fault... Check Ixxx.x / Ixxx.x German' | French: 'S5 904 Row 91 Switch Fault... Check Ixxx.x / Ixxx.x French'
  905 = 'Spare' | German: 'S5 905 Row 91 Spare Message German' | French: 'S5 905 Row 91 Spare Message French'
  906 = 'Spare' | German: 'S5 906 Row 91 Spare Message German' | French: 'S5 906 Row 91 Spare Message French'
  907 = 'Spare' | German: 'S5 907 Row 91 Spare Message German' | French: 'S5 907 Row 91 Spare Message French'
  908 = 'Spare' | German: 'S5 908 Row 91 Spare Message German' | French: 'S5 908 Row 91 Spare Message French'
  909 = 'Spare' | German: 'S5 909 Row 91 Spare Message German' | French: 'S5 909 Row 91 Spare Message French'
  910 = 'Clamp Cylinder A1 Failed to Advance... Check Q1.0...' | German: 'S5 910 Row 92 Failed To Advance.. Check Qxxx.x German' | French: 'S5 910 Row 92 Failed To Advance.. Check Qxxx.x French'
  911 = 'Clamp Cylinder A1 Failed to Return... Check Q1.1...' | German: 'S5 911 Row 92 Failed To Return.. Check Qxxx.x German' | French: 'S5 911 Row 92 Failed To Return.. Check Qxxx.x French'
  912 = 'Clamp Cylinder A1 Lost Advanced... Check I1.0...' | German: 'S5 912 Row 92 Lost Advance Position... Check Ixxx.x German' | French: 'S5 912 Row 92 Lost Advance Position... Check Ixxx.x French'
  913 = 'Clamp Cylinder A1 Lost Returned... Check I1.1...' | German: 'S5 913 Row 92 Lost Return Position... Check Ixxx.x German' | French: 'S5 913 Row 92 Lost Return Position... Check Ixxx.x French'
  914 = 'Clamp Cylinder A1 Switch Fault... Check I1.0, I1.1...' | German: 'S5 914 Row 92 Switch Fault... Check Ixxx.x / Ixxx.x German' | French: 'S5 914 Row 92 Switch Fault... Check Ixxx.x / Ixxx.x French'
  915 = 'Spare' | German: 'S5 915 Row 92 Spare Message German' | French: 'S5 915 Row 92 Spare Message French'
  916 = 'Spare' | German: 'S5 916 Row 92 Spare Message German' | French: 'S5 916 Row 92 Spare Message French'
  917 = 'Spare' | German: 'S5 917 Row 92 Spare Message German' | French: 'S5 917 Row 92 Spare Message French'
  918 = 'Spare' | German: 'S5 918 Row 92 Spare Message German' | French: 'S5 918 Row 92 Spare Message French'
  919 = 'Spare' | German: 'S5 919 Row 92 Spare Message German' | French: 'S5 919 Row 92 Spare Message French'
  920 = 'Clamp Cylinder A1 Failed to Advance... Check Q1.0...' | German: 'S5 920 Row 93 Failed To Advance.. Check Qxxx.x German' | French: 'S5 920 Row 93 Failed To Advance.. Check Qxxx.x French'
  921 = 'Clamp Cylinder A1 Failed to Return... Check Q1.1...' | German: 'S5 921 Row 93 Failed To Return.. Check Qxxx.x German' | French: 'S5 921 Row 93 Failed To Return.. Check Qxxx.x French'
  922 = 'Clamp Cylinder A1 Lost Advanced... Check I1.0...' | German: 'S5 922 Row 93 Lost Advance Position... Check Ixxx.x German' | French: 'S5 922 Row 93 Lost Advance Position... Check Ixxx.x French'
  923 = 'Clamp Cylinder A1 Lost Returned... Check I1.1...' | German: 'S5 923 Row 93 Lost Return Position... Check Ixxx.x German' | French: 'S5 923 Row 93 Lost Return Position... Check Ixxx.x French'
  924 = 'Clamp Cylinder A1 Switch Fault... Check I1.0, I1.1...' | German: 'S5 924 Row 93 Switch Fault... Check Ixxx.x / Ixxx.x German' | French: 'S5 924 Row 93 Switch Fault... Check Ixxx.x / Ixxx.x French'
  925 = 'Spare' | German: 'S5 925 Row 93 Spare Message German' | French: 'S5 925 Row 93 Spare Message French'
  926 = 'Spare' | German: 'S5 926 Row 93 Spare Message German' | French: 'S5 926 Row 93 Spare Message French'
  927 = 'Spare' | German: 'S5 927 Row 93 Spare Message German' | French: 'S5 927 Row 93 Spare Message French'
  928 = 'Spare' | German: 'S5 928 Row 93 Spare Message German' | French: 'S5 928 Row 93 Spare Message French'
  929 = 'Spare' | German: 'S5 929 Row 93 Spare Message German' | French: 'S5 929 Row 93 Spare Message French'
  930 = 'Clamp Cylinder A1 Failed to Advance... Check Q1.0...' | German: 'S5 930 Row 94 Failed To Advance.. Check Qxxx.x German' | French: 'S5 930 Row 94 Failed To Advance.. Check Qxxx.x French'
  931 = 'Clamp Cylinder A1 Failed to Return... Check Q1.1...' | German: 'S5 931 Row 94 Failed To Return.. Check Qxxx.x German' | French: 'S5 931 Row 94 Failed To Return.. Check Qxxx.x French'
  932 = 'Clamp Cylinder A1 Lost Advanced... Check I1.0...' | German: 'S5 932 Row 94 Lost Advance Position... Check Ixxx.x German' | French: 'S5 932 Row 94 Lost Advance Position... Check Ixxx.x French'
  933 = 'Clamp Cylinder A1 Lost Returned... Check I1.1...' | German: 'S5 933 Row 94 Lost Return Position... Check Ixxx.x German' | French: 'S5 933 Row 94 Lost Return Position... Check Ixxx.x French'
  934 = 'Clamp Cylinder A1 Switch Fault... Check I1.0, I1.1...' | German: 'S5 934 Row 94 Switch Fault... Check Ixxx.x / Ixxx.x German' | French: 'S5 934 Row 94 Switch Fault... Check Ixxx.x / Ixxx.x French'
  935 = 'Spare' | German: 'S5 935 Row 94 Spare Message German' | French: 'S5 935 Row 94 Spare Message French'
  936 = 'Spare' | German: 'S5 936 Row 94 Spare Message German' | French: 'S5 936 Row 94 Spare Message French'
  937 = 'Spare' | German: 'S5 937 Row 94 Spare Message German' | French: 'S5 937 Row 94 Spare Message French'
  938 = 'Spare' | German: 'S5 938 Row 94 Spare Message German' | French: 'S5 938 Row 94 Spare Message French'
  939 = 'Spare' | German: 'S5 939 Row 94 Spare Message German' | French: 'S5 939 Row 94 Spare Message French'
  940 = 'Clamp Cylinder A1 Failed to Advance... Check Q1.0...' | German: 'S5 940 Row 95 Failed To Advance.. Check Qxxx.x German' | French: 'S5 940 Row 95 Failed To Advance.. Check Qxxx.x French'
  941 = 'Clamp Cylinder A1 Failed to Return... Check Q1.1...' | German: 'S5 941 Row 95 Failed To Return.. Check Qxxx.x German' | French: 'S5 941 Row 95 Failed To Return.. Check Qxxx.x French'
  942 = 'Clamp Cylinder A1 Lost Advanced... Check I1.0...' | German: 'S5 942 Row 95 Lost Advance Position... Check Ixxx.x German' | French: 'S5 942 Row 95 Lost Advance Position... Check Ixxx.x French'
  943 = 'Clamp Cylinder A1 Lost Returned... Check I1.1...' | German: 'S5 943 Row 95 Lost Return Position... Check Ixxx.x German' | French: 'S5 943 Row 95 Lost Return Position... Check Ixxx.x French'
  944 = 'Clamp Cylinder A1 Switch Fault... Check I1.0, I1.1...' | German: 'S5 944 Row 95 Switch Fault... Check Ixxx.x / Ixxx.x German' | French: 'S5 944 Row 95 Switch Fault... Check Ixxx.x / Ixxx.x French'
  945 = 'Spare' | German: 'S5 945 Row 95 Spare Message German' | French: 'S5 945 Row 95 Spare Message French'
  946 = 'Spare' | German: 'S5 946 Row 95 Spare Message German' | French: 'S5 946 Row 95 Spare Message French'
  947 = 'Spare' | German: 'S5 947 Row 95 Spare Message German' | French: 'S5 947 Row 95 Spare Message French'
  948 = 'Spare' | German: 'S5 948 Row 95 Spare Message German' | French: 'S5 948 Row 95 Spare Message French'
  949 = 'Spare' | German: 'S5 949 Row 95 Spare Message German' | French: 'S5 949 Row 95 Spare Message French'
  950 = 'Clamp Cylinder A1 Failed to Advance... Check Q1.0...' | German: 'S5 950 Row 96 Failed To Advance.. Check Qxxx.x German' | French: 'S5 950 Row 96 Failed To Advance.. Check Qxxx.x French'
  951 = 'Clamp Cylinder A1 Failed to Return... Check Q1.1...' | German: 'S5 951 Row 96 Failed To Return.. Check Qxxx.x German' | French: 'S5 951 Row 96 Failed To Return.. Check Qxxx.x French'
  952 = 'Clamp Cylinder A1 Lost Advanced... Check I1.0...' | German: 'S5 952 Row 96 Lost Advance Position... Check Ixxx.x German' | French: 'S5 952 Row 96 Lost Advance Position... Check Ixxx.x French'
  953 = 'Clamp Cylinder A1 Lost Returned... Check I1.1...' | German: 'S5 953 Row 96 Lost Return Position... Check Ixxx.x German' | French: 'S5 953 Row 96 Lost Return Position... Check Ixxx.x French'
  954 = 'Clamp Cylinder A1 Switch Fault... Check I1.0, I1.1...' | German: 'S5 954 Row 96 Switch Fault... Check Ixxx.x / Ixxx.x German' | French: 'S5 954 Row 96 Switch Fault... Check Ixxx.x / Ixxx.x French'
  955 = 'Spare' | German: 'S5 955 Row 96 Spare Message German' | French: 'S5 955 Row 96 Spare Message French'
  956 = 'Spare' | German: 'S5 956 Row 96 Spare Message German' | French: 'S5 956 Row 96 Spare Message French'
  957 = 'Spare' | German: 'S5 957 Row 96 Spare Message German' | French: 'S5 957 Row 96 Spare Message French'
  958 = 'Spare' | German: 'S5 958 Row 96 Spare Message German' | French: 'S5 958 Row 96 Spare Message French'
  959 = 'Spare' | German: 'S5 959 Row 96 Spare Message German' | French: 'S5 959 Row 96 Spare Message French'
  960 = 'Clamp Cylinder A1 Failed to Advance... Check Q1.0...' | German: 'S5 960 Row 97 Failed To Advance.. Check Qxxx.x German' | French: 'S5 960 Row 97 Failed To Advance.. Check Qxxx.x French'
  961 = 'Clamp Cylinder A1 Failed to Return... Check Q1.1...' | German: 'S5 961 Row 97 Failed To Return.. Check Qxxx.x German' | French: 'S5 961 Row 97 Failed To Return.. Check Qxxx.x French'
  962 = 'Clamp Cylinder A1 Lost Advanced... Check I1.0...' | German: 'S5 962 Row 97 Lost Advance Position... Check Ixxx.x German' | French: 'S5 962 Row 97 Lost Advance Position... Check Ixxx.x French'
  963 = 'Clamp Cylinder A1 Lost Returned... Check I1.1...' | German: 'S5 963 Row 97 Lost Return Position... Check Ixxx.x German' | French: 'S5 963 Row 97 Lost Return Position... Check Ixxx.x French'
  964 = 'Clamp Cylinder A1 Switch Fault... Check I1.0, I1.1...' | German: 'S5 964 Row 97 Switch Fault... Check Ixxx.x / Ixxx.x German' | French: 'S5 964 Row 97 Switch Fault... Check Ixxx.x / Ixxx.x French'
  965 = 'Spare' | German: 'S5 965 Row 97 Spare Message German' | French: 'S5 965 Row 97 Spare Message French'
  966 = 'Spare' | German: 'S5 966 Row 97 Spare Message German' | French: 'S5 966 Row 97 Spare Message French'
  967 = 'Spare' | German: 'S5 967 Row 97 Spare Message German' | French: 'S5 967 Row 97 Spare Message French'
  968 = 'Spare' | German: 'S5 968 Row 97 Spare Message German' | French: 'S5 968 Row 97 Spare Message French'
  969 = 'Spare' | German: 'S5 969 Row 97 Spare Message German' | French: 'S5 969 Row 97 Spare Message French'
  970 = 'Clamp Cylinder A1 Failed to Advance... Check Q1.0...' | German: 'S5 970 Row 98 Failed To Advance.. Check Qxxx.x German' | French: 'S5 970 Row 98 Failed To Advance.. Check Qxxx.x French'
  971 = 'Clamp Cylinder A1 Failed to Return... Check Q1.1...' | German: 'S5 971 Row 98 Failed To Return.. Check Qxxx.x German' | French: 'S5 971 Row 98 Failed To Return.. Check Qxxx.x French'
  972 = 'Clamp Cylinder A1 Lost Advanced... Check I1.0...' | German: 'S5 972 Row 98 Lost Advance Position... Check Ixxx.x German' | French: 'S5 972 Row 98 Lost Advance Position... Check Ixxx.x French'
  973 = 'Clamp Cylinder A1 Lost Returned... Check I1.1...' | German: 'S5 973 Row 98 Lost Return Position... Check Ixxx.x German' | French: 'S5 973 Row 98 Lost Return Position... Check Ixxx.x French'
  974 = 'Clamp Cylinder A1 Switch Fault... Check I1.0, I1.1...' | German: 'S5 974 Row 98 Switch Fault... Check Ixxx.x / Ixxx.x German' | French: 'S5 974 Row 98 Switch Fault... Check Ixxx.x / Ixxx.x French'
  975 = 'Spare' | German: 'S5 975 Row 98 Spare Message German' | French: 'S5 975 Row 98 Spare Message French'
  976 = 'Spare' | German: 'S5 976 Row 98 Spare Message German' | French: 'S5 976 Row 98 Spare Message French'
  977 = 'Spare' | German: 'S5 977 Row 98 Spare Message German' | French: 'S5 977 Row 98 Spare Message French'
  978 = 'Spare' | German: 'S5 978 Row 98 Spare Message German' | French: 'S5 978 Row 98 Spare Message French'
  979 = 'Spare' | German: 'S5 979 Row 98 Spare Message German' | French: 'S5 979 Row 98 Spare Message French'
  980 = 'Clamp Cylinder A1 Failed to Advance... Check Q1.0...' | German: 'S5 980 Row 99 Failed To Advance.. Check Qxxx.x German' | French: 'S5 980 Row 99 Failed To Advance.. Check Qxxx.x French'
  981 = 'Clamp Cylinder A1 Failed to Return... Check Q1.1...' | German: 'S5 981 Row 99 Failed To Return.. Check Qxxx.x German' | French: 'S5 981 Row 99 Failed To Return.. Check Qxxx.x French'
  982 = 'Clamp Cylinder A1 Lost Advanced... Check I1.0...' | German: 'S5 982 Row 99 Lost Advance Position... Check Ixxx.x German' | French: 'S5 982 Row 99 Lost Advance Position... Check Ixxx.x French'
  983 = 'Clamp Cylinder A1 Lost Returned... Check I1.1...' | German: 'S5 983 Row 99 Lost Return Position... Check Ixxx.x German' | French: 'S5 983 Row 99 Lost Return Position... Check Ixxx.x French'
  984 = 'Clamp Cylinder A1 Switch Fault... Check I1.0, I1.1...' | German: 'S5 984 Row 99 Switch Fault... Check Ixxx.x / Ixxx.x German' | French: 'S5 984 Row 99 Switch Fault... Check Ixxx.x / Ixxx.x French'
  985 = 'Spare' | German: 'S5 985 Row 99 Spare Message German' | French: 'S5 985 Row 99 Spare Message French'
  986 = 'Spare' | German: 'S5 986 Row 99 Spare Message German' | French: 'S5 986 Row 99 Spare Message French'
  987 = 'Spare' | German: 'S5 987 Row 99 Spare Message German' | French: 'S5 987 Row 99 Spare Message French'
  988 = 'Spare' | German: 'S5 988 Row 99 Spare Message German' | French: 'S5 988 Row 99 Spare Message French'
  989 = 'Spare' | German: 'S5 989 Row 99 Spare Message German' | French: 'S5 989 Row 99 Spare Message French'
  990 = 'S5 990 Row 100 Failed To Advance.. Check Qxxx.x Default' | German: 'S5 990 Row 100 Failed To Advance.. Check Qxxx.x German' | French: 'S5 990 Row 100 Failed To Advance.. Check Qxxx.x French'
  991 = 'S5 991 Row 100 Failed To Return.. Check Qxxx.x Default' | German: 'S5 991 Row 100 Failed To Return.. Check Qxxx.x German' | French: 'S5 991 Row 100 Failed To Return.. Check Qxxx.x French'
  992 = 'S5 992 Row 100 Lost Advance Position... Check Ixxx.x Default' | German: 'S5 992 Row 100 Lost Advance Position... Check Ixxx.x German' | French: 'S5 992 Row 100 Lost Advance Position... Check Ixxx.x French'
  993 = 'S5 993 Row 100 Lost Return Position... Check Ixxx.x Default' | German: 'S5 993 Row 100 Lost Return Position... Check Ixxx.x German' | French: 'S5 993 Row 100 Lost Return Position... Check Ixxx.x French'
  994 = 'S5 994 Row 100 Switch Fault... Check Ixxx.x / Ixxx.x Default' | German: 'S5 994 Row 100 Switch Fault... Check Ixxx.x / Ixxx.x German' | French: 'S5 994 Row 100 Switch Fault... Check Ixxx.x / Ixxx.x French'
  995 = 'S5 995 Row 100 Spare Message Default' | German: 'S5 995 Row 100 Spare Message German' | French: 'S5 995 Row 100 Spare Message French'
  996 = 'S5 996 Row 100 Spare Message Default' | German: 'S5 996 Row 100 Spare Message German' | French: 'S5 996 Row 100 Spare Message French'
  997 = 'S5 997 Row 100 Spare Message Default' | German: 'S5 997 Row 100 Spare Message German' | French: 'S5 997 Row 100 Spare Message French'
  998 = 'S5 998 Row 100 Spare Message Default' | German: 'S5 998 Row 100 Spare Message German' | French: 'S5 998 Row 100 Spare Message French'
  999 = 'S5 999 Row 100 Spare Message Default' | German: 'S5 999 Row 100 Spare Message German' | French: 'S5 999 Row 100 Spare Message French'
  1000 = 'S5_Alarms Default 1000' | German: 'S5_Alarms German 1000' | French: 'S5_Alarms French 1000'
   = ''
END_TEXTLIST

(* stored: Version 1.1.0.1, ProductVersion 3.1.4024.12
   TextList S5_Alarms: Id {45a0465e-7688-4a63-93cf-6473a0aa50da} *)
